{attribute 'qualified_only'}
VAR_GLOBAL CONSTANT
  //Defect manager library constants max array size
  nDefectTableStrLen_C        : UINT := 40;
	nMaxDefects_C    		        : UINT := 1000;
	nMaxDefectsView_C           : UINT := 40;
  tInfoOffTimeout_C           : TIME := T#5S; 
  tInfoOffAndNotAckTimeout_C  : TIME := T#15S;
END_VAR

(* stored: Version 1.1.0.1, ProductVersion 3.1.4024.13
   GVL CDefect: Id {b637d4a5-b39c-4bf9-8f55-3f1254518ed6} *)
